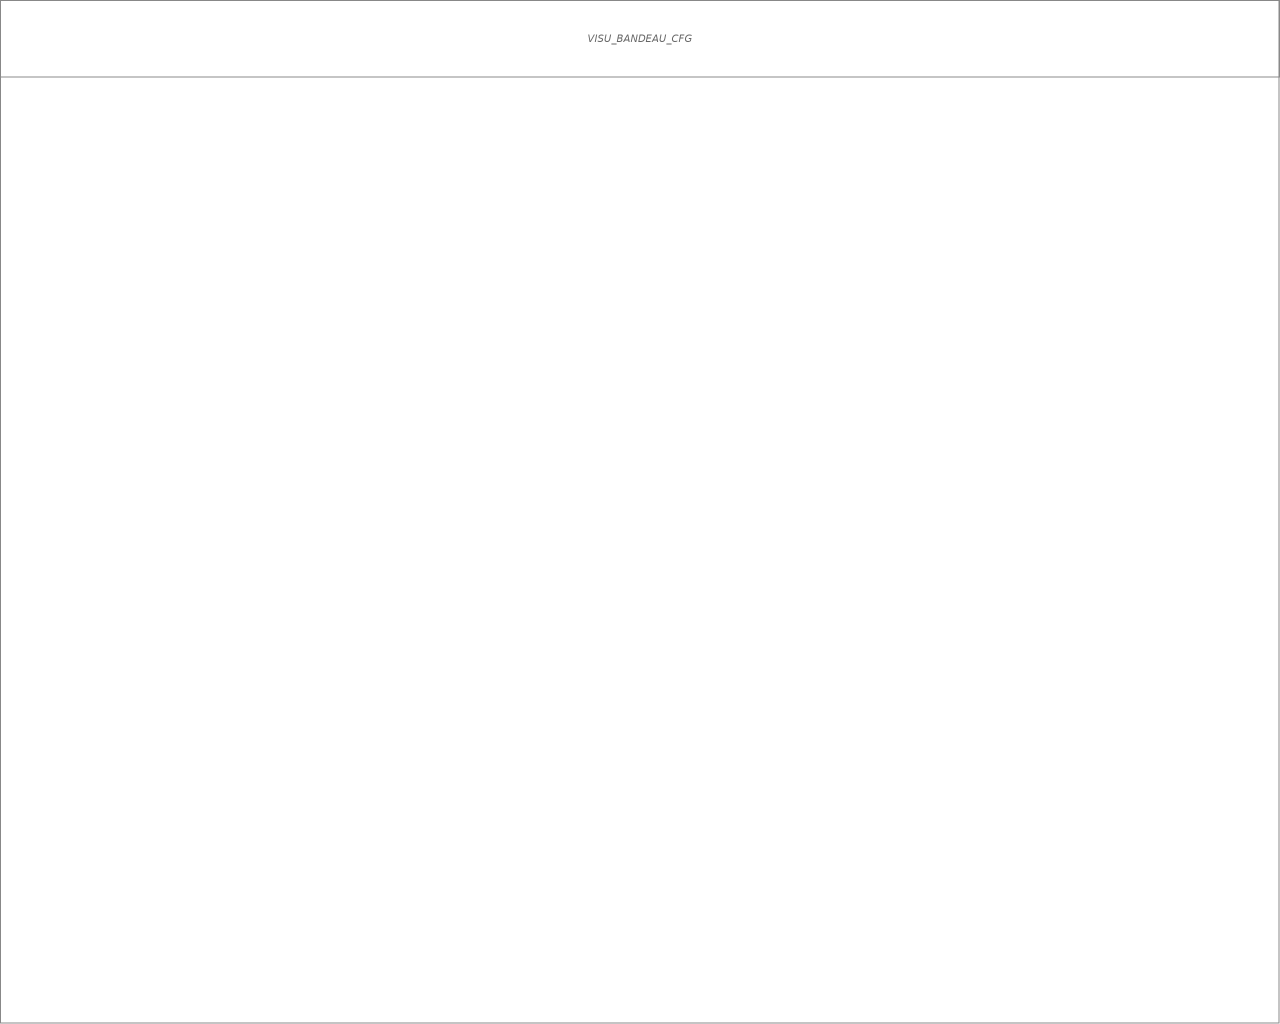
VISUALIZATION VISU_CONFIG_MOUVEMENTS  // 1280x1024, background image fond_blanc_1280_1024
    Frame (0,0 1280x77)
        shows VISU_BANDEAU_CFG()
END_VISUALIZATION

(* stored: Version 1.1.0.1, ProductVersion 3.1.4024.10
   Visu VISU_CONFIG_MOUVEMENTS: Id {26c9ef53-f8f6-4767-8967-862f6484059c} *)
